(* IEC 61131-3 sources: Std_PalletMover/Class/PerPiviotWeel, 1 file *)

(* ---- PerPiviotWeel.st ---- *)
(*!
<Class
	Name               = "PerPiviotWeel"
	Revision           = "0.0"
	RealtimeTask       = "false"
	CyclicTask         = "false"
	BackgroundTask     = "false"
	Sigmatek           = "false"
	OSInterface        = "false"
	HighPriority       = "false"
	Automatic          = "false"
	UpdateMode         = "Prescan"
	SharedCommandTable = "true"
	Objectsize         = "(1260,120)">
	<Channels>
		<Server Name="ClassSvr" Visualized="false" Initialize="false" WriteProtected="true" Retentive="false"/>
		<Server Name="PiviotInterface" Class="I_PivotWheel" Visualized="false" Initialize="false" WriteProtected="true" Retentive="false"/>
		<Server Name="ToObject" Class="CntrlPeriperalPiviotWheels" Visualized="false" Initialize="false" WriteProtected="true" Retentive="false" Comment="ToObject:&#13;&#10;Object channel server.&#13;&#10;Channel to reach the methodes of this object.&#13;&#10;&#13;&#10;In case this object should be Accessible by a pointer&#13;&#10;the variable ToObject is used to handover the address of this object.&#13;&#10;&#13;&#10;This server is never used for anything else!!!&#13;&#10;&#13;&#10;&#13;&#10;"/>
		<Client Name="Curtis_AC2F_IO2_steer" Required="true" Internal="true"/>
		<Client Name="EncoderPulses" Required="false" Internal="false"/>
		<Client Name="Merker1" Required="true" Internal="true"/>
		<Client Name="Obj_Curtis_AC2F_IO2_drive" Required="true" Internal="true"/>
		<Client Name="ObjCurtisDrive" Required="true" Internal="true"/>
		<Client Name="ObjCurtisSteer" Required="true" Internal="true"/>
		<Client Name="ObjDrive" Required="true" Internal="true"/>
		<Client Name="ObjEncoderpulsesToDegrees" Required="true" Internal="true"/>
		<Client Name="ObjPeriperalPiviotWheels" Required="true" Internal="true"/>
		<Client Name="ObjPW" Required="true" Internal="true"/>
		<Client Name="ObjSteer" Required="true" Internal="true"/>
		<Client Name="p_NextObject" Required="false" Internal="false" Comment="Pointer to next object in linked list"/>
		<Client Name="SafetyEncoderValue" Required="true" Internal="false"/>
		<Client Name="SpeedCalculator" Required="true" Internal="true"/>
		<Client Name="ToAgvConfig" Required="true" Internal="false"/>
		<Client Name="ToAgvSettings" Required="true" Internal="false"/>
	</Channels>
	<Network Name="PerPiviotWeel">
		<!-- List of Components in this network -->
		<Components>
			<Object
				Name       = "Curtis_AC2F_IO2_steer"
				Class      = "Curtis_AC2F_IO"
				Position   = "(120,330)"
				Visualized = "true">
				<Channels>
					<Server Name="ClassSvr"/>
					<Server Name="In11_Enc1_c"/>
					<Server Name="In12"/>
					<Server Name="In13"/>
					<Server Name="In14_An14"/>
					<Server Name="In1_An1"/>
					<Server Name="In2_An2_Temp"/>
					<Server Name="In5_An5"/>
					<Server Name="In6_An6"/>
					<Server Name="In7_An7"/>
					<Server Name="In8_An8"/>
					<Server Name="Out1_In21"/>
					<Server Name="Out2_In22"/>
					<Server Name="Out3_In23"/>
					<Server Name="Out4_In24"/>
					<Server Name="Out5_In25"/>
					<Server Name="Out_ResetEm"/>
					<Server Name="xIn21"/>
					<Server Name="xIn22"/>
					<Server Name="xIn23"/>
					<Server Name="xIn24"/>
					<Server Name="xIn25"/>
				</Channels>
			</Object>
			<Object
				Name       = "Merker1"
				Class      = "Merker"
				Position   = "(3390,630)"
				Visualized = "true"
				Remotely   = "true">
				<Channels>
					<Server Name="Data"/>
				</Channels>
			</Object>
			<Object
				Name       = "Obj_Curtis_AC2F_IO2_drive"
				Class      = "Curtis_AC2F_IO"
				Position   = "(150,4080)"
				Visualized = "true">
				<Channels>
					<Server Name="ClassSvr"/>
					<Server Name="In11_Enc1_c"/>
					<Server Name="In12"/>
					<Server Name="In13"/>
					<Server Name="In14_An14"/>
					<Server Name="In1_An1"/>
					<Server Name="In2_An2_Temp"/>
					<Server Name="In5_An5"/>
					<Server Name="In6_An6"/>
					<Server Name="In7_An7"/>
					<Server Name="In8_An8"/>
					<Server Name="Out1_In21"/>
					<Server Name="Out2_In22"/>
					<Server Name="Out3_In23"/>
					<Server Name="Out4_In24"/>
					<Server Name="Out5_In25"/>
					<Server Name="Out_ResetEm"/>
					<Server Name="xIn21"/>
					<Server Name="xIn22"/>
					<Server Name="xIn23"/>
					<Server Name="xIn24"/>
					<Server Name="xIn25"/>
				</Channels>
			</Object>
			<Object
				Name       = "ObjCurtisDrive"
				Class      = "Curtis_AC2F"
				Position   = "(1410,3900)"
				Visualized = "true"
				CyclicTime = "5 ms">
				<Channels>
					<Server Name="Active"/>
					<Server Name="AI_BrakePot"/>
					<Server Name="AI_ThrottlePot"/>
					<Server Name="AutoAccelTime" Value="50"/>
					<Server Name="AutoAct"/>
					<Server Name="AutoDecelTime" Value="10"/>
					<Server Name="AutomaticSetpoint"/>
					<Server Name="AutoSetp"/>
					<Server Name="BDI"/>
					<Server Name="BrakePotSigned"/>
					<Server Name="BusyReferencing"/>
					<Server Name="Capacitor_Voltage"/>
					<Server Name="ClassSvr"/>
					<Server Name="CommunicationOk"/>
					<Server Name="DriveMode"/>
					<Server Name="DriveModeRequest"/>
					<Server Name="EMStop_DiagCode"/>
					<Server Name="EmStopOk"/>
					<Server Name="Enabled" Value="1"/>
					<Server Name="EncoderValue"/>
					<Server Name="Eq_DiagCode"/>
					<Server Name="Fault"/>
					<Server Name="FaultCode"/>
					<Server Name="I_DigitalOut6"/>
					<Server Name="I_DigitalOut7"/>
					<Server Name="I_Driver1"/>
					<Server Name="I_Driver2"/>
					<Server Name="I_Driver3"/>
					<Server Name="I_Driver4"/>
					<Server Name="I_PropDriver"/>
					<Server Name="I_Switch1"/>
					<Server Name="I_Switch16"/>
					<Server Name="I_Switch2"/>
					<Server Name="I_Switch3"/>
					<Server Name="I_Switch4"/>
					<Server Name="I_Switch5"/>
					<Server Name="I_Switch6"/>
					<Server Name="I_Switch7"/>
					<Server Name="I_Switch8"/>
					<Server Name="InterlockExternal1"/>
					<Server Name="InterlockExternal2"/>
					<Server Name="InterlockFeedback"/>
					<Server Name="MonitorValue"/>
					<Server Name="MotorCurrent"/>
					<Server Name="MotorRPM"/>
					<Server Name="MotorTemperature"/>
					<Server Name="ParameterMonitorCase"/>
					<Server Name="ParameterValue"/>
					<Server Name="QD_DigitalOut6"/>
					<Server Name="QD_DigitalOut7"/>
					<Server Name="QD_Driver1"/>
					<Server Name="QD_Driver2"/>
					<Server Name="QD_Driver3"/>
					<Server Name="QD_Driver4"/>
					<Server Name="QD_PropDriver"/>
					<Server Name="Referenced"/>
					<Server Name="ReleaseBrake"/>
					<Server Name="ThrottlePotSigned"/>
					<Client Name="AlarmStartId" Value="1200"/>
					<Client Name="Interlock"/>
					<Client Name="NodeId" Value="1"/>
					<Client Name="objCurtis_AC2F_IO" Value="0"/>
					<Client Name="objDriver" Value="0"/>
					<Client Name="ReleaseBrakesRequest"/>
				</Channels>
			</Object>
			<Object
				Name       = "ObjCurtisSteer"
				Class      = "Curtis_AC2F"
				Position   = "(1410,120)"
				Visualized = "true"
				CyclicTime = "5 ms">
				<Channels>
					<Server Name="Active"/>
					<Server Name="AI_BrakePot"/>
					<Server Name="AI_ThrottlePot"/>
					<Server Name="AutoAccelTime" Value="100"/>
					<Server Name="AutoAct"/>
					<Server Name="AutoDecelTime" Value="10"/>
					<Server Name="AutomaticSetpoint"/>
					<Server Name="AutoSetp"/>
					<Server Name="BDI"/>
					<Server Name="BrakePotSigned"/>
					<Server Name="BusyReferencing"/>
					<Server Name="Capacitor_Voltage"/>
					<Server Name="ClassSvr"/>
					<Server Name="CommunicationOk"/>
					<Server Name="DriveMode"/>
					<Server Name="DriveModeRequest"/>
					<Server Name="EMStop_DiagCode"/>
					<Server Name="EmStopOk"/>
					<Server Name="Enabled" Value="1"/>
					<Server Name="EncoderValue"/>
					<Server Name="Eq_DiagCode"/>
					<Server Name="Fault"/>
					<Server Name="FaultCode"/>
					<Server Name="I_DigitalOut6"/>
					<Server Name="I_DigitalOut7"/>
					<Server Name="I_Driver1"/>
					<Server Name="I_Driver2"/>
					<Server Name="I_Driver3"/>
					<Server Name="I_Driver4"/>
					<Server Name="I_PropDriver"/>
					<Server Name="I_Switch1"/>
					<Server Name="I_Switch16"/>
					<Server Name="I_Switch2"/>
					<Server Name="I_Switch3"/>
					<Server Name="I_Switch4"/>
					<Server Name="I_Switch5"/>
					<Server Name="I_Switch6"/>
					<Server Name="I_Switch7"/>
					<Server Name="I_Switch8"/>
					<Server Name="InterlockExternal1"/>
					<Server Name="InterlockExternal2"/>
					<Server Name="InterlockFeedback"/>
					<Server Name="MonitorValue"/>
					<Server Name="MotorCurrent"/>
					<Server Name="MotorRPM"/>
					<Server Name="MotorTemperature"/>
					<Server Name="ParameterMonitorCase"/>
					<Server Name="ParameterValue"/>
					<Server Name="QD_DigitalOut6"/>
					<Server Name="QD_DigitalOut7"/>
					<Server Name="QD_Driver1"/>
					<Server Name="QD_Driver2"/>
					<Server Name="QD_Driver3"/>
					<Server Name="QD_Driver4"/>
					<Server Name="QD_PropDriver"/>
					<Server Name="Referenced"/>
					<Server Name="ReleaseBrake"/>
					<Server Name="ThrottlePotSigned"/>
					<Client Name="AlarmStartId" Value="1100"/>
					<Client Name="Interlock"/>
					<Client Name="NodeId" Value="2"/>
					<Client Name="objCurtis_AC2F_IO" Value="0"/>
					<Client Name="objDriver" Value="0"/>
					<Client Name="ReleaseBrakesRequest"/>
				</Channels>
			</Object>
			<Object
				Name       = "ObjDrive"
				Class      = "HandleSteeringCurtisAC2F"
				Position   = "(3090,3630)"
				Visualized = "false"
				CyclicTime = "100 ms">
				<Channels>
					<Server Name="Actual"/>
					<Server Name="BusyReferencing"/>
					<Server Name="ClassSvr"/>
					<Server Name="CorrectedActual"/>
					<Server Name="IsReferenced"/>
					<Server Name="ReferenceOffset"/>
					<Server Name="ScalingFactor" Value="-3642.25"/>
					<Server Name="Setpoint"/>
					<Server Name="STARTREF"/>
					<Client Name="ActualRaw"/>
					<Client Name="objCurtisAC2F"/>
					<Client Name="SafetyEncoderValue" Value="0"/>
					<Client Name="SetpointRaw"/>
				</Channels>
			</Object>
			<Object
				Name       = "ObjEncoderpulsesToDegrees"
				Class      = "EncoderpulsesToDegrees"
				Position   = "(2550,540)"
				Visualized = "false"
				CyclicTime = "100 ms">
				<Channels>
					<Server Name="ClassSvr"/>
					<Server Name="Degrees"/>
					<Server Name="GearRatio" Value="4.057"/>
					<Server Name="PulsesPerRound" Value="8192"/>
					<Client Name="EncoderPulses"/>
				</Channels>
			</Object>
			<Object
				Name       = "ObjPeriperalPiviotWheels"
				Class      = "CntrlPeriperalPiviotWheels"
				Position   = "(4200,1050)"
				Visualized = "false">
				<Channels>
					<Server Name="ToObject"/>
					<Client Name="op_LogData"/>
					<Client Name="p_NextObject"/>
					<Client Name="ToAgvConfig"/>
					<Client Name="ToAgvSettings"/>
				</Channels>
			</Object>
			<Object
				Name       = "ObjPW"
				Class      = "I_PivotWheel"
				Position   = "(4200,690)"
				Visualized = "false">
				<Channels>
					<Server Name="ClassSvr"/>
					<Server Name="DistanceToCenterX" Value="2179.966"/>
					<Server Name="DistanceToCenterY" Value="896.5"/>
					<Server Name="PivotWheelReferenced"/>
					<Client Name="objDrive"/>
					<Client Name="objSteer" Value="0"/>
				</Channels>
			</Object>
			<Object
				Name       = "ObjSteer"
				Class      = "HandleSteeringCurtisAC2F"
				Position   = "(3240,300)"
				Visualized = "false"
				CyclicTime = "100 ms">
				<Channels>
					<Server Name="Actual"/>
					<Server Name="BusyReferencing"/>
					<Server Name="ClassSvr"/>
					<Server Name="CorrectedActual"/>
					<Server Name="IsReferenced"/>
					<Server Name="ReferenceOffset"/>
					<Server Name="ScalingFactor" Value="-50"/>
					<Server Name="Setpoint"/>
					<Server Name="STARTREF"/>
					<Client Name="ActualRaw"/>
					<Client Name="objCurtisAC2F"/>
					<Client Name="SafetyEncoderValue"/>
					<Client Name="SetpointRaw"/>
				</Channels>
			</Object>
			<Object
				Name       = "SpeedCalculator"
				Class      = "SpeedCalculator"
				Position   = "(3090,4500)"
				Visualized = "false"
				CyclicTime = "1000 ms">
				<Channels>
					<Server Name="ClassSvr"/>
					<Server Name="mms"/>
					<Client Name="SafetyPulsjes"/>
				</Channels>
			</Object>
		</Components>
		<Comments>
		</Comments>
		<!-- List of Connections in this network -->
		<Connections>
			<Connection Source="this.Merker1" Destination="Merker1.Data"/>
			<Connection Source="this.SpeedCalculator" Destination="SpeedCalculator.ClassSvr"/>
			<Connection Source="this.Curtis_AC2F_IO2_steer" Destination="Curtis_AC2F_IO2_steer.ClassSvr"/>
			<Connection Source="this.ObjPW" Destination="ObjPW.ClassSvr"/>
			<Connection Source="this.ObjCurtisSteer" Destination="ObjCurtisSteer.ClassSvr"/>
			<Connection Source="this.ObjSteer" Destination="ObjSteer.ClassSvr"/>
			<Connection Source="this.ObjEncoderpulsesToDegrees" Destination="ObjEncoderpulsesToDegrees.ClassSvr"/>
			<Connection Source="this.Obj_Curtis_AC2F_IO2_drive" Destination="Obj_Curtis_AC2F_IO2_drive.ClassSvr"/>
			<Connection Source="this.ObjDrive" Destination="ObjDrive.ClassSvr"/>
			<Connection Source="this.ObjCurtisDrive" Destination="ObjCurtisDrive.ClassSvr"/>
			<Connection Source="ObjSteer.SetpointRaw" Destination="ObjCurtisSteer.AutomaticSetpoint" Vertices="(3240,570),(2176,2490),"/>
			<Connection Source="ObjSteer.objCurtisAC2F" Destination="ObjCurtisSteer.ClassSvr" Vertices="(3240,390),(2700,390),(2700,210),(2176,210),"/>
			<Connection Source="ObjDrive.objCurtisAC2F" Destination="ObjCurtisDrive.ClassSvr" Vertices="(3090,3720),(2400,3720),(2400,3930),(2176,3990),"/>
			<Connection Source="ObjSteer.ActualRaw" Destination="ObjCurtisSteer.EncoderValue" Vertices="(3240,510),(2520,510),(2520,3450),(2176,3450),"/>
			<Connection Source="ObjDrive.ActualRaw" Destination="ObjCurtisDrive.MotorRPM" Vertices="(3090,3840),(2490,3840),(2490,5910),(2176,5970),"/>
			<Connection Source="ObjCurtisDrive.objDriver" Destination="CanDriverCPU1.Command"/>
			<Connection Source="ObjDrive.SetpointRaw" Destination="ObjCurtisDrive.AutomaticSetpoint" Vertices="(3090,3900),(2580,3900),(2580,6210),(2176,6270),"/>
			<Connection Source="ObjCurtisSteer.objCurtis_AC2F_IO" Destination="Curtis_AC2F_IO2_steer.ClassSvr" Vertices="(1410,390),(706,420),"/>
			<Connection Source="ObjCurtisDrive.objCurtis_AC2F_IO" Destination="Obj_Curtis_AC2F_IO2_drive.ClassSvr" Vertices="(1410,4170),(736,4170),"/>
			<Connection Source="ObjCurtisSteer.objDriver" Destination="CanDriverCPU1.Command"/>
			<Connection Source="ObjSteer.SafetyEncoderValue" Destination="ObjEncoderpulsesToDegrees.Degrees" Vertices="(3240,450),(3078,810),"/>
			<Connection Source="ObjPW.objSteer" Destination="ObjSteer.ClassSvr" Vertices="(4200,780),(3886,390),"/>
			<Connection Source="ObjPW.objDrive" Destination="ObjDrive.ClassSvr" Vertices="(4200,840),(3736,3720),"/>
			<Connection Source="this.ObjPeriperalPiviotWheels" Destination="ObjPeriperalPiviotWheels.ToObject"/>
			<Connection Source="ObjPeriperalPiviotWheels.p_NextObject" Destination="this.p_NextObject" Vertices="(4200,1200),(38,330),"/>
			<Connection Source="this.ToObject" Destination="ObjPeriperalPiviotWheels.ToObject" Vertices="(5138,330),(4966,1140),"/>
			<Connection Source="ObjEncoderpulsesToDegrees.EncoderPulses" Destination="this.EncoderPulses" Vertices="(2550,630),(38,210),"/>
			<Connection Source="this.PiviotInterface" Destination="ObjPW.ClassSvr" Vertices="(5138,270),(4966,780),"/>
			<Connection Source="ObjDrive.SafetyEncoderValue" Destination="this.SafetyEncoderValue" Vertices="(3090,3780),(38,270),"/>
			<Connection Source="ObjPeriperalPiviotWheels.ToAgvConfig" Destination="this.ToAgvConfig" Vertices="(4200,1260),(38,390),"/>
			<Connection Source="ObjPeriperalPiviotWheels.ToAgvSettings" Destination="this.ToAgvSettings" Vertices="(4200,1320),(38,450),"/>
		</Connections>
		<!-- Headerfiles -->
		<Options>
		</Options>
	</Network>
</Class>
*)
PerPiviotWeel : CLASS
  //Servers:
	ClassSvr 	: SvrChCmd_DINT;
	PiviotInterface 	: SvrChCmd_DINT;
	ToObject 	: SvrChCmd_pVoid;
  //Clients:
	Merker1 	: CltChCmd_Merker;
	ObjCurtisSteer 	: CltChCmd_Curtis_AC2F;
	ObjCurtisDrive 	: CltChCmd_Curtis_AC2F;
	ObjDrive 	: CltChCmd_HandleSteeringCurtisAC2F;
	SpeedCalculator 	: CltChCmd_SpeedCalculator;
	Obj_Curtis_AC2F_IO2_drive 	: CltChCmd_Curtis_AC2F_IO;
	Curtis_AC2F_IO2_steer 	: CltChCmd_Curtis_AC2F_IO;
	ObjPW 	: CltChCmd_I_PivotWheel;
	ObjSteer 	: CltChCmd_HandleSteeringCurtisAC2F;
	ObjEncoderpulsesToDegrees 	: CltChCmd_EncoderpulsesToDegrees;
	EncoderPulses 	: CltCh_DINT;
	SafetyEncoderValue 	: CltCh_REAL;
	ObjPeriperalPiviotWheels 	: CltChCmd_CntrlPeriperalPiviotWheels;
	p_NextObject 	: CltChCmd_LinkedObjectBase;
	ToAgvConfig 	: CltChCmd_AgvConfig;
	ToAgvSettings 	: CltChCmd_AgvSettings;
  //Variables:
  //Functions:

	FUNCTION VIRTUAL GLOBAL PiviotInterface::Read
		VAR_OUTPUT
			output (EAX) 	: DINT;
		END_VAR;

	FUNCTION VIRTUAL GLOBAL ToObject::Read
		VAR_OUTPUT
			output (EAX) 	: pVoid;
		END_VAR;
  //Tables:
	FUNCTION @STD
		VAR_OUTPUT
			ret_code	: CONFSTATES;
		END_VAR;
	FUNCTION GLOBAL TAB @CT_;
END_CLASS;

#pragma using CntrlPeriperalPiviotWheels
#pragma using Curtis_AC2F
#pragma using Curtis_AC2F_IO
#pragma using EncoderpulsesToDegrees
#pragma using HandleSteeringCurtisAC2F
#pragma using I_PivotWheel
#pragma using Merker
#pragma using SpeedCalculator
#pragma usingLtd AgvConfig
#pragma usingLtd AgvSettings
#pragma usingLtd LinkedObjectBase

FUNCTION VIRTUAL GLOBAL PerPiviotWeel::PiviotInterface::Read
	VAR_OUTPUT
		output (EAX) 	: DINT;
	END_VAR

	PiviotInterface := ObjPW.ClassSvr.Read();
	output := PiviotInterface;

END_FUNCTION

FUNCTION VIRTUAL GLOBAL PerPiviotWeel::ToObject::Read
	VAR_OUTPUT
		output (EAX) 	: pVoid;
	END_VAR

	ToObject := ObjPeriperalPiviotWheels.ToObject.Read();
	output := ToObject;

END_FUNCTION
